(********************* G.D S.p.A. - Technical Department ***********************************
This program has been generated automatically from Application Designer DE&F
********************************************************************************************)
PROGRAM dbg_csp_case_feed_magazine_level_zone2
VAR
  di_shd : digital_input_shadow;
END_VAR

_objects_manager();

IF	g_application_status <> APPLICATION_STATUS_RUNNING
THEN
	RETURN;
END_IF

CASE process_get_mode(CONVERSION_this := dbg_root.prc) OF
	MODE_ABSENT,
	MODE_INACTIVE:
		RETURN;
	MODE_TEST:
		RETURN;
END_CASE

ACTION _objects_manager:
IF	objects_initialization()
THEN
	digital_input_shadow_init(
		sim_mode:= SHADOW_SIMULATION_MODE_AUTOMATIC, 
		father:= csp_case_feed_magazine_level_zone2.di, 
		process:= dbg_root.prc, 
		CONVERSION_this:= di_shd);

	RETURN;
END_IF

IF	objects_running()
THEN
	digital_input_shadow_cycle(di_shd);
END_IF
END_ACTION

END_PROGRAM

(* stored: Version 1.1.0.1, ProductVersion 3.1.4022.12
   POU dbg_csp_case_feed_magazine_level_zone2: Id {c83949ec-95f9-417b-9791-ecf0f056dead}, SpecialFunc None
   Action _objects_manager: Id {33042726-d240-4202-acb1-8f68d0c08ffe} *)
